(* CoDeSys 2.3 export: ST_DE_CYLINDER_POS_CFG.EXP *)

(* Data type *)
TYPE ST_DE_CYLINDER_POS_CFG :
STRUCT
	TgtLS_In  : REAL;
	TgtLS_Out : REAL;
	TgtLS_Mid : REAL;
	TgtLS_DB  : REAL;

	LS_Limit_In  : BOOL;
	LS_Limit_Out : BOOL;

	Cycle   : REAL; (*Seconds*)
	TimeMax : REAL; (*Seconds*)

	HP : BYTE;
END_STRUCT
END_TYPE
